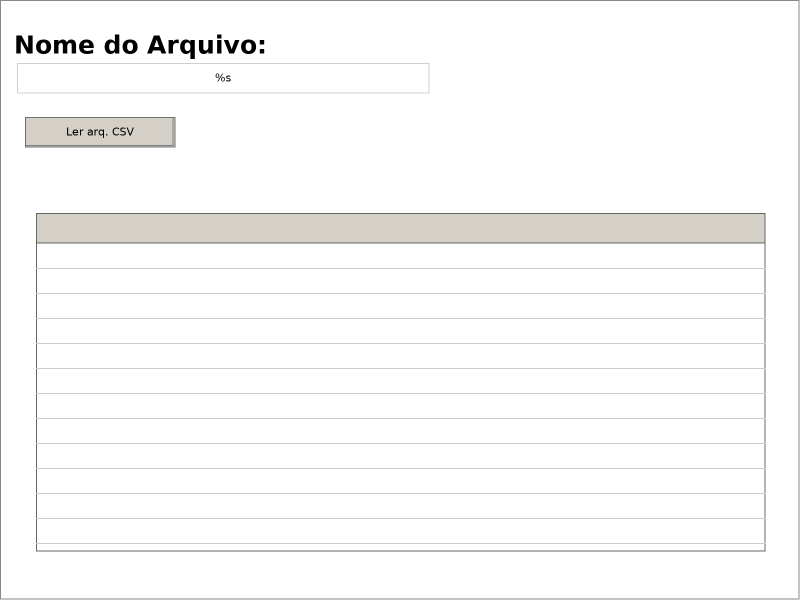
VISUALIZATION Visualization  // 800x600
    Textfield (17,63 412x30), "%s", text variable: MAIN.myNomeArquivo
        OnMouseEnter: write the text variable via Edit
    Label (11,16 377x57), "Nome do Arquivo:"
    Table (36,213 729x338), data array: MAIN.ArrayVisuDB
        p3854506369: MAIN.ArrayVisuDB[0,INDEX]
        p1892666644: MAIN.ArrayVisuDB[1,INDEX]
        p338671338: MAIN.ArrayVisuDB[2,INDEX]
        p2170511999: MAIN.ArrayVisuDB[3,INDEX]
        p3723444502: MAIN.ArrayVisuDB[4,INDEX]
        p1218418051: MAIN.ArrayVisuDB[5,INDEX]
        p746581629: MAIN.ArrayVisuDB[6,INDEX]
        p3104783080: MAIN.ArrayVisuDB[7,INDEX]
        p2501879983: MAIN.ArrayVisuDB[8,INDEX]
        p7306298: MAIN.ArrayVisuDB[9,INDEX]
        p1933151965: MAIN.ArrayVisuDB[10,INDEX]
    Button (25,117 150x30), "Ler arq. CSV"
        tap MAIN.bLer
END_VISUALIZATION

(* stored: Version 1.1.0.1, ProductVersion 3.1.4024.11
   Visu Visualization: Id {44aee93f-8d0a-4fab-8870-65fd9313b0cb} *)
